RoboDK station: UR5e_Endowrist_TCP_orientation.rdk

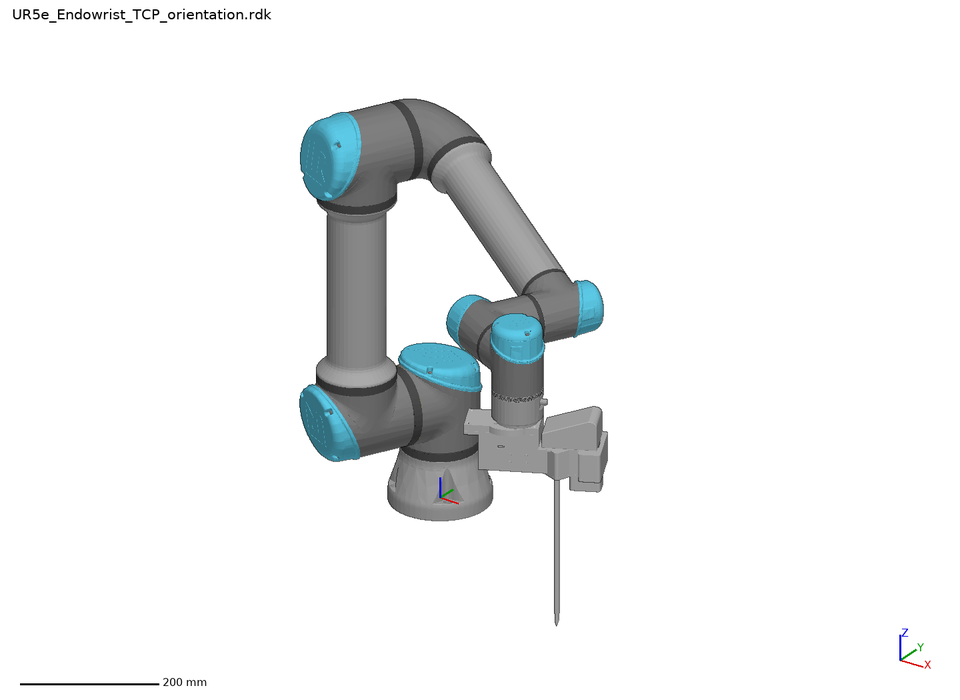
[picture v0: the station drawn from its stored meshes, robots at their saved joint values, targets as dots, program paths as lines]
Station UR5e_Endowrist_TCP_orientation (saved by RoboDK 5.3.0). Poses are relative to the parent item; angles as X-Y-Z fixed-axis rotations.
  - frame UR5e Base at (0, 0, 0) mm
    - robot UR5e: 6 axes, payload 5 kg, reach 850 mm, repeatability 0.03 mm, weight 18.4 kg
        modified DH rows (alpha deg, a mm, theta deg, d mm): 0, 0, 0, 162.5; 90, 0, 180, 0; 0, 425, 0, 0; 0, 392.25, 0, 133.3; -90, 0, 0, 99.7; 90, 0, 180, 99.6
        joint limits [-360, -360, -360, -360, -360, -360] to [360, 360, 360, 360, 360, 360]; home [0, -90, -90, 0, 90, 0]; saved at [-26.14, -90.259, -109.191, -70.535, 90.017, -53.207]
      - tool TCP_Endowrist, TCP at (0, -60, 320) mm, rotated rx -179.74 ry -11.08 rz 53.84 deg, size 82.3 x 200.6 x 341 mm, geometry from Endowrist_TOTAL.stl
  - Python program IMU_controlled_endowrist (listed below)

--- Python program IMU_controlled_endowrist ---
"""
********************************************************************************
RoboticsUB-TCP_Endowrist_from_IMU.py - Control based on a IMU.
Copyright (C) 2021  Albert Álvarez-Carulla
Repository: https://github.com/TheAlbertDev/pcb-esp32-imu

This program is free software: you can redistribute it and/or modify
it under the terms of the GNU General Public License as published by
the Free Software Foundation, either version 3 of the License, or
(at your option) any later version.

This program is distributed in the hope that it will be useful,
but WITHOUT ANY WARRANTY; without even the implied warranty of
MERCHANTABILITY or FITNESS FOR A PARTICULAR PURPOSE.  See the
GNU General Public License for more details.

You should have received a copy of the GNU General Public License
along with this program.  If not, see <https://www.gnu.org/licenses/>.
********************************************************************************
"""

import serial
import time
import math
from enum import Enum

# RoboDK API: import the robolink library (bridge with RoboDK)
from robolink import *
# Robot toolbox: import the robodk library (robotics toolbox)
from robodk import *

# ------------------------------------------------------------------------------
# Connection
# ------------------------------------------------------------------------------

# Establish the connection on a specific port
arduino = serial.Serial('/dev/cu.usbserial-0001', 115200, timeout=1)

# Lets bring some time to the system to stablish the connetction
time.sleep(2)

# Establish a link with the simulator
RDK = Robolink()

# ------------------------------------------------------------------------------
# Simulator setup
# ------------------------------------------------------------------------------

# Retrieve all items (object in the robodk tree)
# Define the "robot" variable with our robot (UR5e)
robot = RDK.Item('UR5e')

# Define the "tcp" variable with the TCP of Endowrist needle
tcp_tool = RDK.Item('TCP_Endowrist')

# Performs a quick check to validate items defined
if robot.Valid():
    print('Robot selected: ' + robot.Name())
if tcp_tool.Valid():
    print('Tool selected: ' + tcp_tool.Name())

# Robot Flange with respect to UR5e base Frame
print('Robot POSE is: ' + repr(robot.Pose()))
# Tool frame with respect to Robot Flange
print('Robot POSE is: ' + repr(robot.PoseTool()))
# Tool frame with respect to Tool frame
print('TCP pose is: ' + repr(tcp_tool.Pose()))

robot.setSpeed(10)

# ------------------------------------------------------------------------------
# Reference frame is fixed to TCP
#
# Data comunication
# ------------------------------------------------------------------------------
#


class Command(Enum):
    GET_RPW = b'\x01'
    GET_QUAT = b'\x02'


try:

    # Discard initial ESP32 message
    arduino.reset_input_buffer()

    while True:

        # Requesting data to Ardino
        arduino.write(Command.GET_RPW.value)

        # Storing received data
        roll_str = arduino.readline().strip()
        pitch_str = arduino.readline().strip()
        yaw_str = arduino.readline().strip()
        torque_str = arduino.readline().strip()
        s1_str = arduino.readline().strip()
        s2_str = arduino.readline().strip()

        # Convert variable values from string to float
        roll = float(roll_str)
        pitch = float(pitch_str)
        yaw = float(yaw_str)
        torque = float(torque_str)
        s1 = bool(int(s1_str))
        s2 = bool(int(s2_str))

        print(roll, pitch, yaw, torque, s1, s2)

        # Convert from degrees to radians R,P,Y angles
        R = math.radians(roll)
        P = math.radians(pitch)
        W = math.radians(yaw)
        X = 0
        Y = -60
        Z = 320

        # Calculate the POSE matrix (UR)
        pose_matrix = transl([X, Y, Z])*rotz(-W)*roty(-P)*rotx(R)*rotx(pi)

        tcp_tool_pose = tcp_tool.setPoseTool(pose_matrix)
        # print ('Tool TCP pose is: ' + repr([R,P,Y]) + '\n')
        # print('Torke Endowrist is: ' + repr([torque]) + '\n')

        approach = robot.Pose()

        if not s1:
            approach = robot.Pose()*transl(0, 10, 0)
            robot.MoveL(approach, False)
        elif not s2:
            approach = robot.Pose()*transl(0, -10, 0)
            robot.MoveL(approach, False)

except KeyboardInterrupt:
    print("Communication stopped.")
    pass

# ------------------------------------------------------------------------------
# Disconnect Arduino
# ------------------------------------------------------------------------------
print("Disconnecting Arduino...")
arduino.close()
